# B&R Automation Studio project SpindleTest
Automation Studio 4.12.5.95 SP; technology packages: mappCockpit 5.24.3, mappMotion 5.27.1, mappView 5.24.4

## Configuration Config1

CPU X20CP0484-1, AutomationRuntime M4.93, Build 4.1.2, Safety 0.0, Vc V4.72.6

### Task classes (Cpu.sw)
```
Cyclic#4 (cycle 100000 us, tolerance 100000 us):
  Program <- Program.prg
Libraries: McBase, MpBase, MpAxis, McAxis, McAcpAx, McDS402Ax, CoTrace, AsZip, FileIO, runtime
```

### Hardware
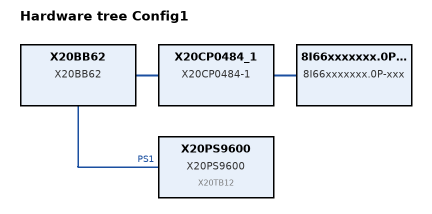
```
8I66xxxxxxx.0P-xxx : 8I66xxxxxxx.0P-xxx v2.6.0.0  [PLK1 -> X20CP0484_1.IF3 (NodeNumber=3) [Cable Type=PowerlinkCable, Length=10, Version=1.0.0.3]]
  FunctionModel = MotionConfig
  McTypeID = McAcoposInverterP66P
  AxisReference = gAxis_1
  InputIsReadOnly = 0
  Input = 1
  OutputIsReadOnly = 0
  Output = 1
  ReferenceDistanceIsReadOnly = 0
  ReferenceDistance = 1
  UnitOfSetpoint = Rpm
  IOM_AIDP1 = LCR
  IOM_AIDP2 = OTR
  IOM_AIDP3 = RFR_D
  IOM_AIDP4 = LFT
  Sel_NameplateMask = 8Ix6T400075_IEC
  Cfg_NSP = 2880
  Cfg_UNS = 380
  Cfg_NCR = 17
  Cfg_COS = 87
X20BB62 : X20BB62 v1.3.0.0
X20CP0484_1 : X20CP0484-1 v1.8.1.0  [SL -> X20BB62.SL1]
  Connector IF2:
    ActivateDevice = 1
    Mode = Manual
    InternetAddress = 192.168.1.182
    SubnetMask = 255.255.255.0
  ConfigurationID = SpindleTest_Config1
  TimerDeviceType = SWIOTIMER
  Cyclic1Duration = 10000
  Cyclic1Tolerance = 10000
  Cyclic2Duration = 20000
  Cyclic2Tolerance = 20000
  Cyclic3Duration = 50000
  Cyclic3Tolerance = 50000
  Cyclic4Duration = 100000
  Cyclic4Tolerance = 100000
  Cyclic5Duration = 200000
  Cyclic5Tolerance = 200000
  Cyclic6Duration = 500000
  Cyclic6Tolerance = 500000
  Cyclic7Duration = 1000000
  Cyclic7Tolerance = 1000000
  Cyclic8Duration = 10000
  Cyclic8Tolerance = 30000000
  FileDevice1
  FileDeviceName1 = USER
  FileDevicePath1 = USER_PATH
  ActivateOpcUa = 1
  OpcUaInformationModels_PV_Version = 1
X20PS9600 : X20PS9600 v1.6.1.0  [PS -> X20BB62.PS1; SS1 -> X20TB12.SS]
X20TB12 : X20TB12 v1.0.0.0
```

### Config_1.axis - X20CP0484_1/mappMotion/Config_1.axis
```
Element gAxis_1 (Type=axis)
  BaseTypeIsReadOnly = 0
  BaseType = Linear
    MeasurementUnit = 5066068
    MeasurementResolutionIsReadOnly = 0
    MeasurementResolution = 1
    CountDirectionIsReadOnly = 0
    CountDirection = Standard
  MovementLimitsIsReadOnly = 0
  MovementLimits = Internal
    Position:
      LowerLimitMin = -1.79769313486231E308
      UpperLimitMax = 1.79769313486231E308
      LowerLimit = -1000.0
      UpperLimit = 1000.0
    VelocityIsReadOnly = 0
    Velocity:
      VelocityMax = 3.4E38
      Velocity = 10.0
    AccelerationIsReadOnly = 0
    Acceleration:
      AccelerationMax = 3.4E38
      Acceleration = 50.0
    DecelerationIsReadOnly = 0
    Deceleration:
      DecelerationMax = 3.4E38
      Deceleration = 50.0
  Alarms = None
```

## Logical view

Binary libraries used (declarations not repeated): operator, runtime, astime, AsIecCon, McBase, MpBase, MpAxis, McAxis, McAcpAx, McDS402Ax 5.27.1, CoTrace, AsZip, FileIO


### Program Logical/Program (IEC)

#### Main.st
```iecst
PROGRAM _INIT
	(* Insert code here *)
	 gAxis_1;

END_PROGRAM

PROGRAM _CYCLIC
	(* Insert code here *)

END_PROGRAM

PROGRAM _EXIT
	(* Insert code here *)

END_PROGRAM
```

Listed in the project but not available here: Logical/Global.typ, Logical/Global.var
